// TIA Portal V20 export
FUNCTION "PostProcess_Send" : Void   // FC2, FBD
{ S7_Optimized_Access := 'TRUE' }
// stored: SetENOAutomatically false
BEGIN

REGION Network 1
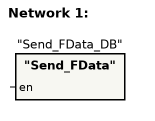
   "Send_FData_DB"();   // "Send_FData"
END_REGION
END_FUNCTION
